(* CODESYS project Ex1.project

Project tree, tasks and I/O mapping:
  Device : CODESYS Control Win V3, 3S - Smart Software Solutions GmbH, order no. 305021, version 3.5.11.30
    application Application
      libraries: Standard, * (System)
      task MainTask (cyclic, interval t#20ms, priority 1) calls PLC_PRG
      program PLC_PRG [ST]
*)

// Device/Application/PLC_PRG
PROGRAM PLC_PRG
VAR
	START : BOOL;
	STOP : BOOL;
	AUX1 : BOOL;
	MV1 : BOOL;
	LT2 :  BOOL;
	MOTOR : BOOL;
	LT3: BOOL;
	T1: TOF;
	T2: TOF;
	AUX2: BOOL;
	TIME1: TIME;
	TIME2: TIME;
	CONT: WORD;
	STIR: BOOL;
	AUX3: BOOL;
	CT1: CTU;
	Q1: BOOL;
	Q2: BOOL;
	R1: R_TRIG;
	R2: R_TRIG;
	MV2: BOOL;
	LT1: BOOL;
END_VAR

IF START THEN 
	AUX1 := TRUE;
END_IF

IF STOP THEN 
	AUX1 := FALSE;
	AUX1 := FALSE;
	MV1 := FALSE;
	MOTOR := FALSE;
	MV2:=FALSE;
END_IF

IF AUX1 THEN 
	MV1 := TRUE;
	
	IF LT2 THEN 
		MV1 := FALSE;
		LT3 := FALSE;
		MOTOR := TRUE;
	END_IF
	IF LT3 THEN 
		LT2 := FALSE;
		MOTOR := FALSE;
		AUX2 := TRUE;
	END_IF
	
	T1(IN:=(R1.Q OR R2.Q) AND NOT(CT1.Q), PT:=T#15S, ET=>TIME1, Q=>Q1);
	T2(IN:=Q1, PT:=T#10S, ET=>TIME2, Q=>Q2);
	
	CT1(CU:=NOT(Q2), RESET:=START OR STOP OR LT1, PV:=3, CV =>CONT);
	
	IF (Q1) THEN
		STIR:=TRUE;
	ELSE
		STIR:=FALSE;
	END_IF
	
	IF CT1.Q THEN 
		MV2:=TRUE;
	END_IF
	
	IF LT1 THEN 
		AUX2 := FALSE;
		MV2:=FALSE;
		MV1:=TRUE;
	END_IF
	
END_IF

R1(CLK:=AUX2);
R2(CLK:=NOT(Q2));

END_PROGRAM
